// Mitsubishi GX Works2 project: 수위제어풀이2   PLC: Q02/Q02H

PROGRAM MAIN
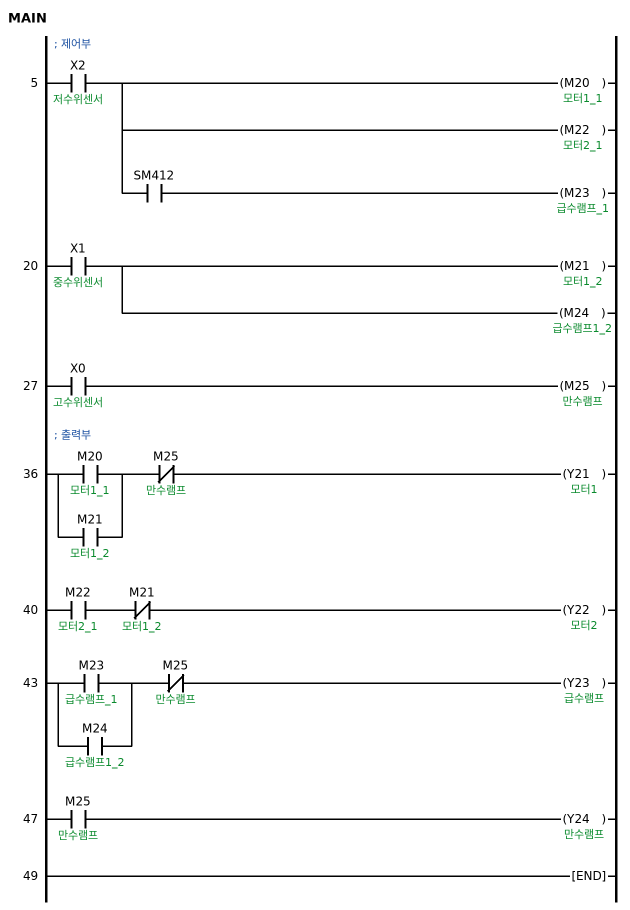
; 제어부
5     LD      X2  ; 저수위센서
      OUT     M20  ; 모터1_1
        [note] 
      OUT     M22  ; 모터2_1
        [note] 모터2_1
      AND     SM412
      OUT     M23  ; 급수램프_1
        [note] 
20    LD      X1  ; 중수위센서
      OUT     M21  ; 모터1_2
        [note] 
      OUT     M24  ; 급수램프1_2
        [note] 
27    LD      X0  ; 고수위센서
      OUT     M25  ; 만수램프
        [note] 
; 출력부
36    LD      M20  ; 모터1_1
      OR      M21  ; 모터1_2
      ANI     M25  ; 만수램프
      OUT     Y21  ; 모터1
40    LD      M22  ; 모터2_1
      ANI     M21  ; 모터1_2
      OUT     Y22  ; 모터2
43    LD      M23  ; 급수램프_1
      OR      M24  ; 급수램프1_2
      ANI     M25  ; 만수램프
      OUT     Y23  ; 급수램프
47    LD      M25  ; 만수램프
      OUT     Y24  ; 만수램프
49    END
END_PROGRAM

// device comments not shown above
M0  ; 보조0
M1  ; 보조1
M2  ; 보조2
M3  ; 보조3
